FUNCTION_BLOCK Conveyor
  (* Standard: 61499-2 *)
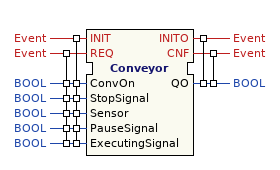
  EVENT_INPUT
    INIT WITH ConvOn, StopSignal, Sensor, PauseSignal, ExecutingSignal;
    REQ WITH ConvOn, StopSignal, Sensor, PauseSignal, ExecutingSignal;
  END_EVENT
  EVENT_OUTPUT
    INITO WITH QO;
    CNF WITH QO;
  END_EVENT
  VAR_INPUT
    ConvOn : BOOL;
    StopSignal : BOOL;
    Sensor : BOOL;
    PauseSignal : BOOL;
    ExecutingSignal : BOOL;
  END_VAR
  VAR_OUTPUT
    QO : BOOL;
  END_VAR
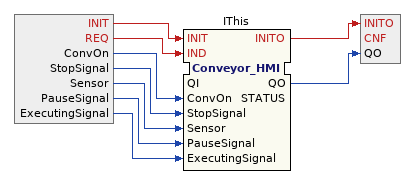
  FBS
    IThis : Conveyor_HMI;
  END_FBS
  EVENT_CONNECTIONS
    INIT TO IThis.INIT;
    REQ TO IThis.IND;
    IThis.INITO TO INITO;
  END_CONNECTIONS
  DATA_CONNECTIONS
    ConvOn TO IThis.ConvOn;
    IThis.QO TO QO;
    StopSignal TO IThis.StopSignal;
    Sensor TO IThis.Sensor;
    PauseSignal TO IThis.PauseSignal;
    ExecutingSignal TO IThis.ExecutingSignal;
  END_CONNECTIONS
END_FUNCTION_BLOCK
